FUNCTION_BLOCK QWStr (* Modbus TCP Client Coil Write Function Block *)
  (* Standard: IEC 61499-1 *)
  (* Version 1.0, AN, SWDC RTSoft *)
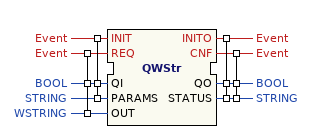
  EVENT_INPUT
    INIT WITH QI, PARAMS; (* Service Initialization *)
    REQ WITH QI, OUT; (* Service Request *)
  END_EVENT
  EVENT_OUTPUT
    INITO WITH QO, STATUS; (* Initialization Confirm *)
    CNF WITH QO, STATUS; (* Confirmation of Requested Service *)
  END_EVENT
  VAR_INPUT
    QI : BOOL; (* Event Input Qualifier *)
    PARAMS : STRING; (* Service Parameters *)
    OUT : WSTRING; (* Input data from resource *)
  END_VAR
  VAR_OUTPUT
    QO : BOOL; (* Event Output Qualifier *)
    STATUS : STRING; (* Service Status *)
  END_VAR
END_FUNCTION_BLOCK
